INTERFACE I_ModuleMaster

PROPERTY iHardwarePool : I_HardwarePool
GET
END_GET
END_PROPERTY

PROPERTY iMasterPrintPosition : I_PrintPosition
GET
END_GET
END_PROPERTY

(*
  Register for PU StatusClient
*)
METHOD registerPuStatusClient : BOOL
VAR_INPUT
  sClient       : I_PrintStatusClient;
END_VAR
END_METHOD

METHOD registerPuSubystem : BOOL
VAR_INPUT
  iSubSys      : I_PrintSubsystem;
END_VAR
END_METHOD

END_INTERFACE

(* stored: Version 1.1.0.1, ProductVersion 3.1.4024.11
   Itf I_ModuleMaster: Id {e3346af7-70cf-49a7-8d6a-452eaef53e1a}
   Property iHardwarePool: Id {47e64cef-1ca8-4871-b850-1ca4d0428620}
   Get Get: Id {f59942ad-49a0-416e-9453-ec512e302676}
   Property iMasterPrintPosition: Id {63258569-32dd-4a07-930d-f166b2c99b0d}
   Get Get: Id {7512c7dc-c219-4c9d-af5f-d83988952e9a}
   Method registerPuStatusClient: Id {38ae4bfc-b4e7-49e2-b782-96ab06eea7b9}
   Method registerPuSubystem: Id {fdb3d458-69d7-471b-a835-e1828f79cf85} *)
